KUKA KRL data list: kuka_ros_driver.dat

&ACCESS RVO2
&REL 13769
&PARAM DISKPATH = KRC:\R1\Program\ROS
DEFDAT  KUKA_ROS_DRIVER PUBLIC
EXT  bas (BAS_COMMAND  :IN,REAL  :IN )

GLOBAL INT ROS_InterfaceVersion=2004
; Controls the communication format of the core server communication
; (must match compile of ROS Node.  See #define in kuka_kss_hw_interface.h)
; 1=EKI_COMM_XML, 2=EKI_COMM_BIN
INT ROS_EKI_COMM_MODE=2

INT ROS_Timeout_RLockID=11
INT ROS_Timeout_SLockID=12
GLOBAL INT ROS_RSI_Conn_Flag=115

E6AXIS ROS_Meas_Pos={A1 -106.622528,A2 -31.4800682,A3 -40.7959671,A4 -36.6705093,A5 72.0757370,A6 139.748947,E1 0.0,E2 0.0,E3 0.0,E4 0.0,E5 0.0,E6 0.0}
E6AXIS ROS_Meas_Vel={A1 0.0,A2 0.0,A3 0.0,A4 0.0,A5 0.0,A6 0.0,E1 0.0,E2 0.0,E3 0.0,E4 0.0,E5 0.0,E6 0.0}
E6AXIS ROS_Meas_Torque={A1 0.0,A2 0.0,A3 0.0,A4 0.0,A5 0.0,A6 0.0,E1 0.0,E2 0.0,E3 0.0,E4 0.0,E5 0.0,E6 0.0}

INT ROS_IPOC=747628430
INT IPOC_END=747628432
; Time for next data send, interval (ms) between sends
INT ROS_Interval=20
GLOBAL BOOL ROS_DoSendTrig=TRUE
GLOBAL BOOL ROS_DidInit=FALSE
; Time for next data collect cycle
INT ROS_NextTrigDC=747628450
INT ROS_IntervalDC=20
GLOBAL BOOL ROS_CommFromSPS=TRUE
GLOBAL INT ROS_InterruptRecv=14
GLOBAL INT ROS_InterruptSend=16
INT recv_status=0

; Operation state types
GLOBAL ENUM ROS_OpStateType Unknown,KRL_PTP,RSI4ms_Pos,RSI12ms_Pos,RSI4ms_Vel,RSI12ms_Vel
GLOBAL ENUM ROS_CommandType ROSC_None,ROSC_Init,ROSC_CmdJpos,ROSC_Start,ROSC_Stop,ROSC_Reset,ROSC_DrivesOn,ROSC_DrivesOff,ROSC_Change,ROSC_Heartbeat,ROSC_SInit,ROSC_SInitName,ROSC_SInitMod,ROSC_SInitRobV,ROSC_SjState,ROSC_Sstatus,ROSC_Sackn
GLOBAL STRUC ROS_CommandItem ROS_CommandType type,CHAR IDstr[8],BOOL isRecv
GLOBAL STRUC ROS_Command ROS_CommandType type,INT cmdID,INT dataID,INT t_recv,INT t_exec,INT i_exe
GLOBAL STRUC ROS_PosItem INT cmdIdx,REAL dt,E6AXIS cmdPos
GLOBAL STRUC ROS_OpStateProgAttr ROS_OpStateType type,CHAR IDstr[64],CHAR prgName[64]
GLOBAL STRUC ROS_OpStateItem ROS_OpStateType type,INT t_recv,INT t_active
GLOBAL STRUC ROS_RobStatusType INT statCode,INT mode,eStop,guardStop,drivesPowered,motionPossible,inMotion,inError,errCode,CHAR opState[64]
GLOBAL STRUC ROS_FeatuesType INT EKI,INT RSI,INT MXA
GLOBAL STRUC CircQueue INT size,INT istart,INT iend

DECL ROS_RobStatusType ROS_RobotStatus
DECL ROS_FeatuesType ROS_SupportFeatures

INT OpStateErrCnt=0
INT OpStateChangeStep=0
INT ROS_CurrentOpStateID=1
DECL GLOBAL ROS_OpStateType ROS_CurrentOpState=#KRL_PTP
DECL GLOBAL ROS_OpStateType ROS_RequestedOpState=#KRL_PTP
BOOL ROS_ChangingOpState=FALSE
CHAR ROS_OpStateProg[256]
ROS_OpStateProg[]="ros_krlptp"

DECL ROS_OpStateType temp_PrevOpState=#KRL_PTP
CHAR tempOpState[64]
tempOpState[]="KRL_PTP"
BOOL tempRB=TRUE

DECL ROS_CommandItem ROS_EmptyCommand={type #ROSC_None,IDstr[] "none",isRecv FALSE}
; Registerd command types
INT ROS_NumCommands=16
INT ROS_MaxCommands=20
DECL GLOBAL ROS_CommandItem ROS_CommandTypes[21] ; last item is always none
ROS_CommandTypes[1]={type #ROSC_Init,IDstr[] "Connect-",isRecv TRUE}
ROS_CommandTypes[2]={type #ROSC_CmdJpos,IDstr[] "CmdJpos-",isRecv TRUE}
ROS_CommandTypes[3]={type #ROSC_Start,IDstr[] "Start---",isRecv TRUE}
ROS_CommandTypes[4]={type #ROSC_Stop,IDstr[] "Stop----",isRecv TRUE}
ROS_CommandTypes[5]={type #ROSC_Reset,IDstr[] "Reset---",isRecv TRUE}
ROS_CommandTypes[6]={type #ROSC_DrivesOn,IDstr[] "DriveOn-",isRecv TRUE}
ROS_CommandTypes[7]={type #ROSC_DrivesOff,IDstr[] "DriveOff",isRecv TRUE}
ROS_CommandTypes[8]={type #ROSC_Change,IDstr[] "Change--",isRecv TRUE}
ROS_CommandTypes[9]={type #ROSC_Heartbeat,IDstr[] "HB------",isRecv TRUE}
ROS_CommandTypes[10]={type #ROSC_SInit,IDstr[] "Init----",isRecv FALSE}
ROS_CommandTypes[11]={type #ROSC_SInitName,IDstr[] "InitName",isRecv FALSE}
ROS_CommandTypes[12]={type #ROSC_SInitMod,IDstr[] "InitMod-",isRecv FALSE}
ROS_CommandTypes[13]={type #ROSC_SInitRobV,IDstr[] "InitRobV",isRecv FALSE}
ROS_CommandTypes[14]={type #ROSC_SjState,IDstr[] "JState--",isRecv FALSE}
ROS_CommandTypes[15]={type #ROSC_Sstatus,IDstr[] "Status--",isRecv FALSE}
ROS_CommandTypes[16]={type #ROSC_Sackn,IDstr[] "Ack-----",isRecv FALSE}
ROS_CommandTypes[17]={type #ROSC_None,IDstr[] "none",isRecv FALSE}
ROS_CommandTypes[18]={type #ROSC_None,IDstr[] "none",isRecv FALSE}
ROS_CommandTypes[19]={type #ROSC_None,IDstr[] "none",isRecv FALSE}
ROS_CommandTypes[20]={type #ROSC_None,IDstr[] "none",isRecv FALSE}
ROS_CommandTypes[21]={type #ROSC_None,IDstr[] "none"}
; Quick indexes for send command
GLOBAL INT ROS_Cmd_____Init=10
GLOBAL INT ROS_Cmd_InitName=11
GLOBAL INT ROS_Cmd__InitMod=12
GLOBAL INT ROS_Cmd_InitRobV=13
GLOBAL INT ROS_Cmd___JState=14
GLOBAL INT ROS_Cmd___Status=15
GLOBAL INT ROS_Cmd_____Ackn=16

; This static structure maps between OpState, communication, and KRL program name
INT ROS_NumOpPrograms=6
DECL ROS_OpStateProgAttr ROS_OpPrograms[10]
ROS_OpPrograms[1]={type #KRL_PTP,IDstr[] "KRL_PTP",prgName[] "ros_krlptp"}
ROS_OpPrograms[2]={type #RSI4ms_Pos,IDstr[] "RSI4ms_Pos",prgName[] "ros_rsi_ext"}
ROS_OpPrograms[3]={type #RSI12ms_Pos,IDstr[] "RSI12ms_Pos",prgName[] "ros_rsi_12ms"}
ROS_OpPrograms[4]={type #RSI4ms_Vel,IDstr[] "RSI4ms_Vel",prgName[] "ros_rsi_ext"}
ROS_OpPrograms[5]={type #RSI12ms_Vel,IDstr[] "RSI12ms_Vel",prgName[] "ros_rsi_12ms"}
ROS_OpPrograms[6]={type #Unknown,IDstr[] "Unknown",prgName[] "none"}

; Bit mapping of status code
GLOBAL INT ROSSTAT_T1=1
GLOBAL INT ROSSTAT_T2=2
GLOBAL INT ROSSTAT_AUTO=4
GLOBAL INT ROSSTAT_EXT=8
GLOBAL INT ROSSTAT_Estop=16
GLOBAL INT ROSSTAT_GuardStop=32
GLOBAL INT ROSSTAT_DrivesPwr=64
GLOBAL INT ROSSTAT_MotionPossible=128
GLOBAL INT ROSSTAT_InMotion=256
GLOBAL INT ROSSTAT_KRL_PTP=512
GLOBAL INT ROSSTAT_RSI4ms_Pos=1024
GLOBAL INT ROSSTAT_RSI12ms_Pos=2048
GLOBAL INT ROSSTAT_RSI4ms_Vel=4096
GLOBAL INT ROSSTAT_RSI12ms_Vel=8192
GLOBAL INT ROSSTAT_InError=32768
INT ROSSTAT_Code_ID=1



REAL vel_ratio[12]
vel_ratio[1]=0.233695656
vel_ratio[2]=0.202702701
vel_ratio[3]=0.232432425
vel_ratio[4]=2.12917962E-06
vel_ratio[5]=0.00337662338
vel_ratio[6]=0.134297520
vel_ratio[7]=0.0
vel_ratio[8]=0.0
vel_ratio[9]=0.0
vel_ratio[10]=0.0
vel_ratio[11]=0.0
vel_ratio[12]=0.0

BOOL lock_data_collect=FALSE
BOOL lock_data_read=FALSE

; Test & performance monitoring vars
INT t_DataCollect=35
INT n_DataCollect=17
GLOBAL REAL ROS_DataCollect_cycle=2.05882359

INT t_write=22
INT n_write=7
GLOBAL REAL ROS_write_cycle=0.0
INT dbg_err_idx=10

INT n_lockHoldRead=3300
INT n_lockHoldCollect=7438



DECL ROS_Command emptyCMD={type #ROSC_None,cmdID -1,t_recv 0,t_exec 0}



DECL CircQueue CMDlist_q={size 100,istart 50,iend 50}
DECL ROS_Command CMDlist[100]
CMDlist[1]={type #ROSC_CmdJpos,cmdID 747189637,dataID 97,t_recv 747189704,t_exec 747191325}
CMDlist[2]={type #ROSC_CmdJpos,cmdID 747189664,dataID 98,t_recv 747189730,t_exec 747191409}
CMDlist[3]={type #ROSC_CmdJpos,cmdID 747189692,dataID 99,t_recv 747189757,t_exec 747191493}
CMDlist[4]={type #ROSC_CmdJpos,cmdID 747189720,dataID 100,t_recv 747189784,t_exec 747191577}
CMDlist[5]={type #ROSC_CmdJpos,cmdID 747189747,dataID 1,t_recv 747189812,t_exec 747191661}
CMDlist[6]={type #ROSC_CmdJpos,cmdID 747189774,dataID 2,t_recv 747189840,t_exec 747191745}
CMDlist[7]={type #ROSC_CmdJpos,cmdID 747189800,dataID 3,t_recv 747189870,t_exec 747191829}
CMDlist[8]={type #ROSC_CmdJpos,cmdID 747189829,dataID 4,t_recv 747189898,t_exec 747191925}
CMDlist[9]={type #ROSC_CmdJpos,cmdID 747189858,dataID 5,t_recv 747189923,t_exec 747192009}
CMDlist[10]={type #ROSC_CmdJpos,cmdID 747189887,dataID 6,t_recv 747189950,t_exec 747192093}
CMDlist[11]={type #ROSC_CmdJpos,cmdID 747189913,dataID 7,t_recv 747189975,t_exec 747192177}
CMDlist[12]={type #ROSC_CmdJpos,cmdID 747189940,dataID 8,t_recv 747190023,t_exec 747192273}
CMDlist[13]={type #ROSC_CmdJpos,cmdID 747189965,dataID 9,t_recv 747190030,t_exec 747192357}
CMDlist[14]={type #ROSC_CmdJpos,cmdID 747189992,dataID 10,t_recv 747190059,t_exec 747192441}
CMDlist[15]={type #ROSC_CmdJpos,cmdID 747190012,dataID 11,t_recv 747190087,t_exec 747192537}
CMDlist[16]={type #ROSC_CmdJpos,cmdID 747190049,dataID 12,t_recv 747190114,t_exec 747192621}
CMDlist[17]={type #ROSC_CmdJpos,cmdID 747190076,dataID 13,t_recv 747190141,t_exec 747192705}
CMDlist[18]={type #ROSC_CmdJpos,cmdID 747190104,dataID 14,t_recv 747190168,t_exec 747192789}
CMDlist[19]={type #ROSC_CmdJpos,cmdID 747190131,dataID 15,t_recv 747190195,t_exec 747192873}
CMDlist[20]={type #ROSC_CmdJpos,cmdID 747190158,dataID 16,t_recv 747190225,t_exec 747192957}
CMDlist[21]={type #ROSC_CmdJpos,cmdID 747190185,dataID 17,t_recv 747190251,t_exec 747193053}
CMDlist[22]={type #ROSC_CmdJpos,cmdID 747190214,dataID 18,t_recv 747190280,t_exec 747193137}
CMDlist[23]={type #ROSC_CmdJpos,cmdID 747190241,dataID 19,t_recv 747190307,t_exec 747193233}
CMDlist[24]={type #ROSC_CmdJpos,cmdID 747190269,dataID 20,t_recv 747190351,t_exec 747193329}
CMDlist[25]={type #ROSC_CmdJpos,cmdID 747190297,dataID 21,t_recv 747190358,t_exec 747193425}
CMDlist[26]={type #ROSC_CmdJpos,cmdID 747190324,dataID 22,t_recv 747190392,t_exec 747193521}
CMDlist[27]={type #ROSC_CmdJpos,cmdID 747190368,dataID 23,t_recv 747190429,t_exec 747193617}
CMDlist[28]={type #ROSC_CmdJpos,cmdID 747190403,dataID 24,t_recv 747190465,t_exec 747193713}
CMDlist[29]={type #ROSC_CmdJpos,cmdID 747190438,dataID 25,t_recv 747190501,t_exec 747193809}
CMDlist[30]={type #ROSC_CmdJpos,cmdID 747190475,dataID 26,t_recv 747190534,t_exec 747193905}
CMDlist[31]={type #ROSC_CmdJpos,cmdID 747190510,dataID 27,t_recv 747190567,t_exec 747194013}
CMDlist[32]={type #ROSC_CmdJpos,cmdID 747190544,dataID 28,t_recv 747190603,t_exec 747194133}
CMDlist[33]={type #ROSC_CmdJpos,cmdID 747190578,dataID 29,t_recv 747190640,t_exec 747194241}
CMDlist[34]={type #ROSC_CmdJpos,cmdID 747190614,dataID 30,t_recv 747190676,t_exec 747194361}
CMDlist[35]={type #ROSC_CmdJpos,cmdID 747190650,dataID 31,t_recv 747190712,t_exec 747194481}
CMDlist[36]={type #ROSC_CmdJpos,cmdID 747190687,dataID 32,t_recv 747190747,t_exec 747194601}
CMDlist[37]={type #ROSC_CmdJpos,cmdID 747190723,dataID 33,t_recv 747190780,t_exec 747194733}
CMDlist[38]={type #ROSC_CmdJpos,cmdID 747190757,dataID 34,t_recv 747190816,t_exec 747194853}
CMDlist[39]={type #ROSC_CmdJpos,cmdID 747190790,dataID 35,t_recv 747190852,t_exec 747194973}
CMDlist[40]={type #ROSC_CmdJpos,cmdID 747190825,dataID 36,t_recv 747190888,t_exec 747195093}
CMDlist[41]={type #ROSC_CmdJpos,cmdID 747190862,dataID 37,t_recv 747190923,t_exec 747195201}
CMDlist[42]={type #ROSC_CmdJpos,cmdID 747190897,dataID 38,t_recv 747190957,t_exec 747195321}
CMDlist[43]={type #ROSC_CmdJpos,cmdID 747190932,dataID 39,t_recv 747191020,t_exec 747195417}
CMDlist[44]={type #ROSC_CmdJpos,cmdID 747190967,dataID 40,t_recv 747191027,t_exec 747195513}
CMDlist[45]={type #ROSC_CmdJpos,cmdID 747190992,dataID 41,t_recv 747191064,t_exec 747195597}
CMDlist[46]={type #ROSC_CmdJpos,cmdID 747191038,dataID 42,t_recv 747191100,t_exec 747195681}
CMDlist[47]={type #ROSC_CmdJpos,cmdID 747191074,dataID 43,t_recv 747191135,t_exec 747195753}
CMDlist[48]={type #ROSC_CmdJpos,cmdID 747191110,dataID 44,t_recv 747191171,t_exec 747195837}
CMDlist[49]={type #ROSC_Stop,cmdID 747233232,t_recv 747233291,t_exec 747233305}
CMDlist[50]={type #ROSC_Reset,cmdID 747246081,t_recv 747246134,t_exec 747246143}
CMDlist[51]={type #ROSC_CmdJpos,cmdID 747152086,dataID 47,t_recv 747152148,t_exec 747154473}
CMDlist[52]={type #ROSC_CmdJpos,cmdID 747152112,dataID 48,t_recv 747152173,t_exec 747154533}
CMDlist[53]={type #ROSC_CmdJpos,cmdID 747152138,dataID 49,t_recv 747152202,t_exec 747154605}
CMDlist[54]={type #ROSC_CmdJpos,cmdID 747152163,dataID 50,t_recv 747152231,t_exec 747154653}
CMDlist[55]={type #ROSC_CmdJpos,cmdID 747152190,dataID 51,t_recv 747152261,t_exec 747154713}
CMDlist[56]={type #ROSC_CmdJpos,cmdID 747152220,dataID 52,t_recv 747152290,t_exec 747154773}
CMDlist[57]={type #ROSC_CmdJpos,cmdID 747152249,dataID 53,t_recv 747152317,t_exec 747154821}
CMDlist[58]={type #ROSC_CmdJpos,cmdID 747152278,dataID 54,t_recv 747152343,t_exec 747154857}
CMDlist[59]={type #ROSC_CmdJpos,cmdID 747188462,dataID 55,t_recv 747188514,t_exec 747188516}
CMDlist[60]={type #ROSC_CmdJpos,cmdID 747188491,dataID 56,t_recv 747188546,t_exec 747188548}
CMDlist[61]={type #ROSC_CmdJpos,cmdID 747188523,dataID 57,t_recv 747188579,t_exec 747188582}
CMDlist[62]={type #ROSC_CmdJpos,cmdID 747188555,dataID 58,t_recv 747188613,t_exec 747188733}
CMDlist[63]={type #ROSC_CmdJpos,cmdID 747188588,dataID 59,t_recv 747188650,t_exec 747188757}
CMDlist[64]={type #ROSC_CmdJpos,cmdID 747188625,dataID 60,t_recv 747188684,t_exec 747188781}
CMDlist[65]={type #ROSC_CmdJpos,cmdID 747188659,dataID 61,t_recv 747188716,t_exec 747188817}
CMDlist[66]={type #ROSC_CmdJpos,cmdID 747188693,dataID 62,t_recv 747188749,t_exec 747188853}
CMDlist[67]={type #ROSC_CmdJpos,cmdID 747188725,dataID 63,t_recv 747188790,t_exec 747188889}
CMDlist[68]={type #ROSC_CmdJpos,cmdID 747188759,dataID 64,t_recv 747188797,t_exec 747188937}
CMDlist[69]={type #ROSC_CmdJpos,cmdID 747188759,dataID 65,t_recv 747188826,t_exec 747188985}
CMDlist[70]={type #ROSC_CmdJpos,cmdID 747188780,dataID 66,t_recv 747188857,t_exec 747189033}
CMDlist[71]={type #ROSC_CmdJpos,cmdID 747188815,dataID 67,t_recv 747188884,t_exec 747189093}
CMDlist[72]={type #ROSC_CmdJpos,cmdID 747188846,dataID 68,t_recv 747188911,t_exec 747189153}
CMDlist[73]={type #ROSC_CmdJpos,cmdID 747188874,dataID 69,t_recv 747188936,t_exec 747189213}
CMDlist[74]={type #ROSC_CmdJpos,cmdID 747188901,dataID 70,t_recv 747188962,t_exec 747189273}
CMDlist[75]={type #ROSC_CmdJpos,cmdID 747188926,dataID 71,t_recv 747188989,t_exec 747189333}
CMDlist[76]={type #ROSC_CmdJpos,cmdID 747188952,dataID 72,t_recv 747189018,t_exec 747189405}
CMDlist[77]={type #ROSC_CmdJpos,cmdID 747188978,dataID 73,t_recv 747189046,t_exec 747189477}
CMDlist[78]={type #ROSC_CmdJpos,cmdID 747189007,dataID 74,t_recv 747189075,t_exec 747189537}
CMDlist[79]={type #ROSC_CmdJpos,cmdID 747189036,dataID 75,t_recv 747189103,t_exec 747189609}
CMDlist[80]={type #ROSC_CmdJpos,cmdID 747189063,dataID 76,t_recv 747189130,t_exec 747189681}
CMDlist[81]={type #ROSC_CmdJpos,cmdID 747189092,dataID 77,t_recv 747189155,t_exec 747189753}
CMDlist[82]={type #ROSC_CmdJpos,cmdID 747189119,dataID 78,t_recv 747189181,t_exec 747189825}
CMDlist[83]={type #ROSC_CmdJpos,cmdID 747189145,dataID 79,t_recv 747189211,t_exec 747189899}
CMDlist[84]={type #ROSC_CmdJpos,cmdID 747189171,dataID 80,t_recv 747189238,t_exec 747189969}
CMDlist[85]={type #ROSC_CmdJpos,cmdID 747189199,dataID 81,t_recv 747189266,t_exec 747190053}
CMDlist[86]={type #ROSC_CmdJpos,cmdID 747189227,dataID 82,t_recv 747189294,t_exec 747190125}
CMDlist[87]={type #ROSC_CmdJpos,cmdID 747189254,dataID 83,t_recv 747189323,t_exec 747190197}
CMDlist[88]={type #ROSC_CmdJpos,cmdID 747189282,dataID 84,t_recv 747189350,t_exec 747190281}
CMDlist[89]={type #ROSC_CmdJpos,cmdID 747189311,dataID 85,t_recv 747189377,t_exec 747190353}
CMDlist[90]={type #ROSC_CmdJpos,cmdID 747189340,dataID 86,t_recv 747189404,t_exec 747190425}
CMDlist[91]={type #ROSC_CmdJpos,cmdID 747189367,dataID 87,t_recv 747189431,t_exec 747190509}
CMDlist[92]={type #ROSC_CmdJpos,cmdID 747189392,dataID 88,t_recv 747189459,t_exec 747190593}
CMDlist[93]={type #ROSC_CmdJpos,cmdID 747189420,dataID 89,t_recv 747189486,t_exec 747190677}
CMDlist[94]={type #ROSC_CmdJpos,cmdID 747189448,dataID 90,t_recv 747189514,t_exec 747190749}
CMDlist[95]={type #ROSC_CmdJpos,cmdID 747189475,dataID 91,t_recv 747189541,t_exec 747190833}
CMDlist[96]={type #ROSC_CmdJpos,cmdID 747189503,dataID 92,t_recv 747189566,t_exec 747190917}
CMDlist[97]={type #ROSC_CmdJpos,cmdID 747189530,dataID 93,t_recv 747189591,t_exec 747191001}
CMDlist[98]={type #ROSC_CmdJpos,cmdID 747189556,dataID 94,t_recv 747189621,t_exec 747191073}
CMDlist[99]={type #ROSC_CmdJpos,cmdID 747189581,dataID 95,t_recv 747189648,t_exec 747191157}
CMDlist[100]={type #ROSC_CmdJpos,cmdID 747189609,dataID 96,t_recv 747189676,t_exec 747191241}


GLOBAL E6AXIS g_joint_pos_empty={A1 0.0,A2 0.0,A3 0.0,A4 0.0,A5 0.0,A6 0.0,E1 0.0,E2 0.0,E3 0.0,E4 0.0,E5 0.0,E6 0.0}
GLOBAL E6AXIS ROS_joint_pos_tgt={A1 -106.622528,A2 -31.4800682,A3 -40.7959671,A4 -36.6705093,A5 72.0757370,A6 139.748947,E1 -0.00564089,E2 0.00186683913,E3 0.0,E4 0.0,E5 0.0,E6 0.0}
; Handshake variables to main motion run to avoid running the same point repeatedly
GLOBAL INT ROS_move_ID=747191110
GLOBAL INT ROS_move_ID_previous=387826110
GLOBAL REAL ROS_move_interval=0.0360000
BOOL ROS_move_init=FALSE

BOOL lock_cmdPos_receive=FALSE
BOOL lock_cmdPos_read=FALSE

DECL CircQueue JPosList_q={size 100,istart 44,iend 44}
DECL ROS_PosItem JPos_log[100]
JPos_log[1]={cmdIdx 5,dt 0.0280000,cmdPos {A1 -62.1725273,A2 -55.9574471,A3 7.92842150,A4 15.2566948,A5 9.14249134,A6 139.747818,E1 -0.00282434770,E2 0.000934711075,E3 0.0,E4 0.0,E5 0.0,E6 0.0}}
JPos_log[2]={cmdIdx 6,dt 0.0270000,cmdPos {A1 -63.2651711,A2 -55.3557587,A3 6.73070860,A4 13.9802523,A5 10.6894779,A6 139.747849,E1 -0.00289358222,E2 0.000957624114,E3 0.0,E4 0.0,E5 0.0,E6 0.0}}
JPos_log[3]={cmdIdx 7,dt 0.0270000,cmdPos {A1 -64.3578110,A2 -54.7540703,A3 5.53299570,A4 12.7038097,A5 12.2364635,A6 139.747879,E1 -0.00296281651,E2 0.000980537,E3 0.0,E4 0.0,E5 0.0,E6 0.0}}
JPos_log[4]={cmdIdx 8,dt 0.0260000,cmdPos {A1 -65.4099884,A2 -54.1746674,A3 4.37964249,A4 11.4746428,A5 13.7261543,A6 139.747894,E1 -0.00302948686,E2 0.00100260146,E3 0.0,E4 0.0,E5 0.0,E6 0.0}}
JPos_log[5]={cmdIdx 9,dt 0.0290000,cmdPos {A1 -66.5835648,A2 -53.5284119,A3 3.09321046,A4 10.1036491,A5 15.3877316,A6 139.747925,E1 -0.00310385,E2 0.00102721166,E3 0.0,E4 0.0,E5 0.0,E6 0.0}}
JPos_log[6]={cmdIdx 10,dt 0.0290000,cmdPos {A1 -67.7571487,A2 -52.8821526,A3 1.80677807,A4 8.73265553,A5 17.0493088,A6 139.747955,E1 -0.00317821279,E2 0.00105182198,E3 0.0,E4 0.0,E5 0.0,E6 0.0}}
JPos_log[7]={cmdIdx 11,dt 0.0290000,cmdPos {A1 -68.9307251,A2 -52.2358971,A3 0.520345867,A4 7.36166191,A5 18.7108860,A6 139.747986,E1 -0.00325257587,E2 0.00107643218,E3 0.0,E4 0.0,E5 0.0,E6 0.0}}
JPos_log[8]={cmdIdx 12,dt 0.0260000,cmdPos {A1 -69.9828949,A2 -51.6564941,A3 -0.633007228,A4 6.13249540,A5 20.2005768,A6 139.748016,E1 -0.00331924600,E2 0.00109849661,E3 0.0,E4 0.0,E5 0.0,E6 0.0}}
JPos_log[9]={cmdIdx 13,dt 0.0270000,cmdPos {A1 -71.0755386,A2 -51.0548058,A3 -1.83072007,A4 4.85605288,A5 21.7475624,A6 139.748047,E1 -0.00338848052,E2 0.00112140959,E3 0.0,E4 0.0,E5 0.0,E6 0.0}}
JPos_log[10]={cmdIdx 14,dt 0.0250000,cmdPos {A1 -72.0872498,A2 -50.4976883,A3 -2.93971348,A4 3.67416167,A5 23.1799583,A6 139.748077,E1 -0.00345258671,E2 0.00114262535,E3 0.0,E4 0.0,E5 0.0,E6 0.0}}
JPos_log[11]={cmdIdx 15,dt 0.0270000,cmdPos {A1 -73.1798859,A2 -49.8960,A3 -4.13742638,A4 2.39771938,A5 24.7269440,A6 139.748093,E1 -0.00352182123,E2 0.00116553833,E3 0.0,E4 0.0,E5 0.0,E6 0.0}}
JPos_log[12]={cmdIdx 16,dt 0.0200000,cmdPos {A1 -73.9892502,A2 -49.4503059,A3 -5.02462101,A4 1.45220637,A5 25.8728600,A6 139.748123,E1 -0.00357310590,E2 0.00118251087,E3 0.0,E4 0.0,E5 0.0,E6 0.0}}
JPos_log[13]={cmdIdx 17,dt 0.0370000,cmdPos {A1 -75.4865799,A2 -48.6257706,A3 -6.66593122,A4 -0.296992451,A5 27.9928036,A6 139.748154,E1 -0.00366798276,E2 0.00121391017,E3 0.0,E4 0.0,E5 0.0,E6 0.0}}
JPos_log[14]={cmdIdx 18,dt 0.0270000,cmdPos {A1 -76.5792236,A2 -48.0240822,A3 -7.86364365,A4 -1.57343483,A5 29.5397892,A6 139.748184,E1 -0.00373721728,E2 0.00123682315,E3 0.0,E4 0.0,E5 0.0,E6 0.0}}
JPos_log[15]={cmdIdx 19,dt 0.0280000,cmdPos {A1 -77.7123337,A2 -47.4001083,A3 -9.10571671,A4 -2.89715290,A5 31.1440716,A6 139.748215,E1 -0.00380901620,E2 0.00126058480,E3 0.0,E4 0.0,E5 0.0,E6 0.0}}
JPos_log[16]={cmdIdx 20,dt 0.0270000,cmdPos {A1 -78.8049698,A2 -46.7984200,A3 -10.3034296,A4 -4.17359543,A5 32.6910553,A6 139.748245,E1 -0.00387825072,E2 0.00128349778,E3 0.0,E4 0.0,E5 0.0,E6 0.0}}
JPos_log[17]={cmdIdx 21,dt 0.0270000,cmdPos {A1 -79.8976135,A2 -46.1967316,A3 -11.5011425,A4 -5.45003796,A5 34.2380447,A6 139.748276,E1 -0.00394748524,E2 0.00130641076,E3 0.0,E4 0.0,E5 0.0,E6 0.0}}
JPos_log[18]={cmdIdx 22,dt 0.0270000,cmdPos {A1 -80.9902573,A2 -45.5950470,A3 -12.6988544,A4 -6.72648,A5 35.7850304,A6 139.748291,E1 -0.00401671976,E2 0.00132932374,E3 0.0,E4 0.0,E5 0.0,E6 0.0}}
JPos_log[19]={cmdIdx 23,dt 0.0290000,cmdPos {A1 -82.1638336,A2 -44.9487877,A3 -13.9852867,A4 -8.09747410,A5 37.4466057,A6 139.748322,E1 -0.00409108261,E2 0.00135393406,E3 0.0,E4 0.0,E5 0.0,E6 0.0}}
JPos_log[20]={cmdIdx 24,dt 0.0270000,cmdPos {A1 -83.2564774,A2 -44.3471,A3 -15.1830,A4 -9.37391663,A5 38.9935913,A6 139.748352,E1 -0.00416031713,E2 0.00137684704,E3 0.0,E4 0.0,E5 0.0,E6 0.0}}
JPos_log[21]={cmdIdx 25,dt 0.0280000,cmdPos {A1 -84.3895874,A2 -43.7231293,A3 -16.4250717,A4 -10.6976347,A5 40.5978737,A6 139.748383,E1 -0.00423211604,E2 0.00140060869,E3 0.0,E4 0.0,E5 0.0,E6 0.0}}
JPos_log[22]={cmdIdx 26,dt 0.0280000,cmdPos {A1 -85.5227,A2 -43.0991554,A3 -17.6671448,A4 -12.0213528,A5 42.2021561,A6 139.748413,E1 -0.00430391449,E2 0.00142437033,E3 0.0,E4 0.0,E5 0.0,E6 0.0}}
JPos_log[23]={cmdIdx 27,dt 0.0270000,cmdPos {A1 -86.6153412,A2 -42.4974670,A3 -18.8648586,A4 -13.2977943,A5 43.7491417,A6 139.748444,E1 -0.00437314902,E2 0.00144728331,E3 0.0,E4 0.0,E5 0.0,E6 0.0}}
JPos_log[24]={cmdIdx 28,dt 0.0440000,cmdPos {A1 -88.3959427,A2 -41.5169411,A3 -20.8166866,A4 -15.3779230,A5 46.2701569,A6 139.748489,E1 -0.00448597595,E2 0.00148462295,E3 0.0,E4 0.0,E5 0.0,E6 0.0}}
JPos_log[25]={cmdIdx 29,dt 0.0350000,cmdPos {A1 -89.8123322,A2 -40.7369728,A3 -22.3692760,A4 -17.0325699,A5 48.2755089,A6 139.748520,E1 -0.00457572425,E2 0.00151432503,E3 0.0,E4 0.0,E5 0.0,E6 0.0}}
JPos_log[26]={cmdIdx 30,dt 0.0350000,cmdPos {A1 -91.2287216,A2 -39.9570084,A3 -23.9218674,A4 -18.6872177,A5 50.2808609,A6 139.748550,E1 -0.00466547254,E2 0.00154402701,E3 0.0,E4 0.0,E5 0.0,E6 0.0}}
JPos_log[27]={cmdIdx 31,dt 0.0370000,cmdPos {A1 -92.7260437,A2 -39.1324730,A3 -25.5631771,A4 -20.4364166,A5 52.4008064,A6 139.748596,E1 -0.00476034964,E2 0.00157542631,E3 0.0,E4 0.0,E5 0.0,E6 0.0}}
JPos_log[28]={cmdIdx 32,dt 0.0350000,cmdPos {A1 -94.1424332,A2 -38.3525085,A3 -27.1157684,A4 -22.0910645,A5 54.4061584,A6 139.748627,E1 -0.00485009793,E2 0.00160512840,E3 0.0,E4 0.0,E5 0.0,E6 0.0}}
JPos_log[29]={cmdIdx 33,dt 0.0340000,cmdPos {A1 -95.5351486,A2 -37.5855789,A3 -28.6424103,A4 -23.7180576,A5 56.3779907,A6 139.748672,E1 -0.00493834633,E2 0.00163433398,E3 0.0,E4 0.0,E5 0.0,E6 0.0}}
JPos_log[30]={cmdIdx 34,dt 0.0340000,cmdPos {A1 -96.9221573,A2 -36.8217926,A3 -30.1627922,A4 -25.3383789,A5 58.3417435,A6 139.748703,E1 -0.00502623292,E2 0.00166341977,E3 0.0,E4 0.0,E5 0.0,E6 0.0}}
JPos_log[31]={cmdIdx 35,dt 0.0360000,cmdPos {A1 -98.2725525,A2 -36.0781631,A3 -31.6430511,A4 -26.9159393,A5 60.2536697,A6 139.748734,E1 -0.00511180,E2 0.00169173803,E3 0.0,E4 0.0,E5 0.0,E6 0.0}}
JPos_log[32]={cmdIdx 36,dt 0.0360000,cmdPos {A1 -99.5495300,A2 -35.3749695,A3 -33.0428238,A4 -28.4077244,A5 62.0616417,A6 139.748764,E1 -0.00519271474,E2 0.00171851658,E3 0.0,E4 0.0,E5 0.0,E6 0.0}}
JPos_log[33]={cmdIdx 37,dt 0.0370000,cmdPos {A1 -100.730888,A2 -34.7244301,A3 -34.3377800,A4 -29.7878036,A5 63.7342300,A6 139.748795,E1 -0.00526757073,E2 0.00174329,E3 0.0,E4 0.0,E5 0.0,E6 0.0}}
JPos_log[34]={cmdIdx 38,dt 0.0360000,cmdPos {A1 -101.813744,A2 -34.1281319,A3 -35.5247650,A4 -31.0528107,A5 65.2673569,A6 139.748825,E1 -0.00533618499,E2 0.00176599773,E3 0.0,E4 0.0,E5 0.0,E6 0.0}}
JPos_log[35]={cmdIdx 39,dt 0.0340000,cmdPos {A1 -102.758011,A2 -33.6081467,A3 -36.5598373,A4 -32.1559219,A5 66.6042786,A6 139.748856,E1 -0.00539601827,E2 0.00178579928,E3 0.0,E4 0.0,E5 0.0,E6 0.0}}
JPos_log[36]={cmdIdx 40,dt 0.0330000,cmdPos {A1 -103.485611,A2 -33.2074776,A3 -37.3574028,A4 -33.0059166,A5 67.6344299,A6 139.748871,E1 -0.00544212200,E2 0.00180105725,E3 0.0,E4 0.0,E5 0.0,E6 0.0}}
JPos_log[37]={cmdIdx 41,dt 0.0350000,cmdPos {A1 -104.116714,A2 -32.8599472,A3 -38.0492,A4 -33.7431831,A5 68.5279541,A6 139.748886,E1 -0.00548211113,E2 0.00181429170,E3 0.0,E4 0.0,E5 0.0,E6 0.0}}
JPos_log[38]={cmdIdx 42,dt 0.0370000,cmdPos {A1 -104.720726,A2 -32.5273361,A3 -38.7112923,A4 -34.4488,A5 69.3831329,A6 139.748901,E1 -0.00552038429,E2 0.00182695792,E3 0.0,E4 0.0,E5 0.0,E6 0.0}}
JPos_log[39]={cmdIdx 43,dt 0.0350000,cmdPos {A1 -105.247467,A2 -32.2372742,A3 -39.2886848,A4 -35.0641479,A5 70.1289,A6 139.748917,E1 -0.00555376057,E2 0.00183800387,E3 0.0,E4 0.0,E5 0.0,E6 0.0}}
JPos_log[40]={cmdIdx 44,dt 0.0350000,cmdPos {A1 -105.720406,A2 -31.9768429,A3 -39.8070946,A4 -35.6166344,A5 70.7984924,A6 139.748932,E1 -0.00558372773,E2 0.00184792140,E3 0.0,E4 0.0,E5 0.0,E6 0.0}}
JPos_log[41]={cmdIdx 45,dt 0.0350000,cmdPos {A1 -106.115677,A2 -31.7591763,A3 -40.2403793,A4 -36.0784,A5 71.3581238,A6 139.748932,E1 -0.00560877379,E2 0.00185621041,E3 0.0,E4 0.0,E5 0.0,E6 0.0}}
JPos_log[42]={cmdIdx 46,dt 0.0250000,cmdPos {A1 -106.335602,A2 -31.6380672,A3 -40.4814568,A4 -36.3353233,A5 71.6695,A6 139.748947,E1 -0.00562270964,E2 0.00186082232,E3 0.0,E4 0.0,E5 0.0,E6 0.0}}
JPos_log[43]={cmdIdx 47,dt 0.0460000,cmdPos {A1 -106.578506,A2 -31.5043068,A3 -40.7477188,A4 -36.6190910,A5 72.0134125,A6 139.748947,E1 -0.00563810114,E2 0.00186591607,E3 0.0,E4 0.0,E5 0.0,E6 0.0}}
JPos_log[44]={cmdIdx 48,dt 0.0360000,cmdPos {A1 -106.622528,A2 -31.4800682,A3 -40.7959671,A4 -36.6705093,A5 72.0757370,A6 139.748947,E1 -0.00564089,E2 0.00186683913,E3 0.0,E4 0.0,E5 0.0,E6 0.0}}
JPos_log[45]={cmdIdx 49,dt 0.0260000,cmdPos {A1 -14.3644066,A2 -80.5024490,A3 60.3516808,A4 67.3275833,A5 -53.9648666,A6 139.746643,E1 0.000590378651,E2 -0.00209156843,E3 0.0,E4 0.0,E5 0.0,E6 0.0}}
JPos_log[46]={cmdIdx 50,dt 0.0290000,cmdPos {A1 -15.0494108,A2 -80.5024948,A3 59.5970306,A4 67.3276291,A5 -53.9649277,A6 139.746658,E1 0.000597995764,E2 -0.00211855397,E3 0.0,E4 0.0,E5 0.0,E6 0.0}}
JPos_log[47]={cmdIdx 51,dt 0.0280000,cmdPos {A1 -15.6574450,A2 -80.5025330,A3 58.9271774,A4 67.3276672,A5 -53.9649811,A6 139.746658,E1 0.000604757,E2 -0.00214250735,E3 0.0,E4 0.0,E5 0.0,E6 0.0}}
JPos_log[48]={cmdIdx 52,dt 0.0280000,cmdPos {A1 -16.2008190,A2 -80.5025635,A3 58.3285599,A4 67.3277054,A5 -53.9650269,A6 139.746674,E1 0.000610799179,E2 -0.00216391333,E3 0.0,E4 0.0,E5 0.0,E6 0.0}}
JPos_log[49]={cmdIdx 53,dt 0.0260000,cmdPos {A1 -16.6365185,A2 -80.5025940,A3 57.8485603,A4 67.3277359,A5 -53.9650650,A6 139.746674,E1 0.000615644094,E2 -0.00218107761,E3 0.0,E4 0.0,E5 0.0,E6 0.0}}
JPos_log[50]={cmdIdx 54,dt 0.0260000,cmdPos {A1 -16.9965782,A2 -80.5026169,A3 57.4518929,A4 67.3277588,A5 -53.9651,A6 139.746674,E1 0.000619647850,E2 -0.00219526212,E3 0.0,E4 0.0,E5 0.0,E6 0.0}}
JPos_log[51]={cmdIdx 55,dt 0.0250000,cmdPos {A1 -17.2649841,A2 -80.5026321,A3 57.1562,A4 67.3277740,A5 -53.9651222,A6 139.746674,E1 0.000622632506,E2 -0.00220583589,E3 0.0,E4 0.0,E5 0.0,E6 0.0}}
JPos_log[52]={cmdIdx 56,dt 0.0270000,cmdPos {A1 -17.4654026,A2 -80.5026474,A3 56.9354019,A4 67.3277893,A5 -53.9651375,A6 139.746689,E1 0.000624861103,E2 -0.00221373141,E3 0.0,E4 0.0,E5 0.0,E6 0.0}}
JPos_log[53]={cmdIdx 57,dt 0.0300000,cmdPos {A1 -17.5805531,A2 -80.5026550,A3 56.8085442,A4 67.3278,A5 -53.9651489,A6 139.746689,E1 0.000626141555,E2 -0.00221826765,E3 0.0,E4 0.0,E5 0.0,E6 0.0}}
JPos_log[54]={cmdIdx 58,dt 0.0290000,cmdPos {A1 -17.5993538,A2 -80.5026550,A3 56.7878342,A4 67.3278,A5 -53.9651489,A6 139.746689,E1 0.000626350637,E2 -0.00221900828,E3 0.0,E4 0.0,E5 0.0,E6 0.0}}
JPos_log[55]={cmdIdx 59,dt 0.0310000,cmdPos {A1 -17.6183434,A2 -80.4921951,A3 56.7670174,A4 67.3056183,A5 -53.9382629,A6 139.746689,E1 0.000616256555,E2 -0.00218711211,E3 0.0,E4 0.0,E5 0.0,E6 0.0}}
JPos_log[56]={cmdIdx 60,dt 0.0280000,cmdPos {A1 -17.7043266,A2 -80.4448471,A3 56.6727676,A4 67.2051697,A5 -53.8165283,A6 139.746689,E1 0.000572450052,E2 -0.00204941514,E3 0.0,E4 0.0,E5 0.0,E6 0.0}}
JPos_log[57]={cmdIdx 61,dt 0.0290000,cmdPos {A1 -17.8910942,A2 -80.3420,A3 56.4680405,A4 66.9869843,A5 -53.5520973,A6 139.746689,E1 0.000482904317,E2 -0.00177018612,E3 0.0,E4 0.0,E5 0.0,E6 0.0}}
JPos_log[58]={cmdIdx 62,dt 0.0320000,cmdPos {A1 -18.2141380,A2 -80.1641083,A3 56.1139297,A4 66.6096,A5 -53.0947266,A6 139.746704,E1 0.000341430394,E2 -0.00133472227,E3 0.0,E4 0.0,E5 0.0,E6 0.0}}
JPos_log[59]={cmdIdx 63,dt 0.0320000,cmdPos {A1 -18.6380062,A2 -79.9306946,A3 55.6493034,A4 66.1144257,A5 -52.4946022,A6 139.746719,E1 0.000179555369,E2 -0.000847501564,E3 0.0,E4 0.0,E5 0.0,E6 0.0}}
JPos_log[60]={cmdIdx 64,dt 0.0330000,cmdPos {A1 -19.1446476,A2 -79.6517,A3 55.0939445,A4 65.5225601,A5 -51.7772903,A6 139.746735,E1 2.33041046E-05,E2 -0.000397049676,E3 0.0,E4 0.0,E5 0.0,E6 0.0}}
JPos_log[61]={cmdIdx 65,dt 0.0370000,cmdPos {A1 -19.7553940,A2 -79.3153839,A3 54.4244652,A4 64.8090744,A5 -50.9125824,A6 139.746750,E1 -0.000105858584,E2 -6.37531630E-05,E3 0.0,E4 0.0,E5 0.0,E6 0.0}}
JPos_log[62]={cmdIdx 66,dt 0.0340000,cmdPos {A1 -20.3424530,A2 -78.9921,A3 53.7809525,A4 64.1232681,A5 -50.0814133,A6 139.746765,E1 -0.000172276414,E2 5.20744034E-05,E3 0.0,E4 0.0,E5 0.0,E6 0.0}}
JPos_log[63]={cmdIdx 67,dt 0.0340000,cmdPos {A1 -20.9898243,A2 -78.6356201,A3 53.0713310,A4 63.3669968,A5 -49.1648483,A6 139.746780,E1 -0.000214834727,E2 7.10990425E-05,E3 0.0,E4 0.0,E5 0.0,E6 0.0}}
JPos_log[64]={cmdIdx 68,dt 0.0320000,cmdPos {A1 -21.7620773,A2 -78.2103577,A3 52.2248154,A4 62.4648361,A5 -48.0714760,A6 139.746796,E1 -0.000263768015,E2 8.72933961E-05,E3 0.0,E4 0.0,E5 0.0,E6 0.0}}
JPos_log[65]={cmdIdx 69,dt 0.0340000,cmdPos {A1 -22.7413063,A2 -77.6711273,A3 51.1514206,A4 61.3208847,A5 -46.6850624,A6 139.746826,E1 -0.000325816218,E2 0.000107828098,E3 0.0,E4 0.0,E5 0.0,E6 0.0}}
JPos_log[66]={cmdIdx 70,dt 0.0340000,cmdPos {A1 -23.7676487,A2 -77.1059494,A3 50.0263824,A4 60.1218948,A5 -45.2319450,A6 139.746841,E1 -0.000390849658,E2 0.000129350767,E3 0.0,E4 0.0,E5 0.0,E6 0.0}}
JPos_log[67]={cmdIdx 71,dt 0.0210000,cmdPos {A1 -24.4380360,A2 -76.7367859,A3 49.2915306,A4 59.3387375,A5 -44.2828,A6 139.746857,E1 -0.000433328300,E2 0.000143408965,E3 0.0,E4 0.0,E5 0.0,E6 0.0}}
JPos_log[68]={cmdIdx 72,dt 0.0350000,cmdPos {A1 -25.6592216,A2 -76.0643082,A3 47.9529152,A4 57.9121284,A5 -42.5538177,A6 139.746887,E1 -0.000510707789,E2 0.000169017527,E3 0.0,E4 0.0,E5 0.0,E6 0.0}}
JPos_log[69]={cmdIdx 73,dt 0.0310000,cmdPos {A1 -26.8036633,A2 -75.4341,A3 46.6984215,A4 56.5751724,A5 -40.9334946,A6 139.746918,E1 -0.000583224581,E2 0.000193016778,E3 0.0,E4 0.0,E5 0.0,E6 0.0}}
JPos_log[70]={cmdIdx 74,dt 0.0280000,cmdPos {A1 -27.9015217,A2 -74.8295364,A3 45.4949913,A4 55.2926369,A5 -39.3791237,A6 139.746948,E1 -0.000652789546,E2 0.000216039160,E3 0.0,E4 0.0,E5 0.0,E6 0.0}}
JPos_log[71]={cmdIdx 75,dt 0.0270000,cmdPos {A1 -29.0208912,A2 -74.2131348,A3 44.2679825,A4 53.9849739,A5 -37.7942963,A6 139.746979,E1 -0.000723717618,E2 0.000239512621,E3 0.0,E4 0.0,E5 0.0,E6 0.0}}
JPos_log[72]={cmdIdx 76,dt 0.0250000,cmdPos {A1 -30.0407505,A2 -73.6515274,A3 43.1500511,A4 52.7935562,A5 -36.3503571,A6 139.747009,E1 -0.000788340287,E2 0.000260899338,E3 0.0,E4 0.0,E5 0.0,E6 0.0}}
JPos_log[73]={cmdIdx 77,dt 0.0260000,cmdPos {A1 -31.0929241,A2 -73.0721207,A3 41.9966965,A4 51.5643883,A5 -34.8606682,A6 139.747025,E1 -0.000855010527,E2 0.000282963709,E3 0.0,E4 0.0,E5 0.0,E6 0.0}}
JPos_log[74]={cmdIdx 78,dt 0.0260000,cmdPos {A1 -32.1451,A2 -72.4927139,A3 40.8433456,A4 50.3352242,A5 -33.3709755,A6 139.747055,E1 -0.000921680825,E2 0.000305028050,E3 0.0,E4 0.0,E5 0.0,E6 0.0}}
JPos_log[75]={cmdIdx 79,dt 0.0290000,cmdPos {A1 -33.3186760,A2 -71.8464584,A3 39.5569115,A4 48.9642296,A5 -31.7094,A6 139.747086,E1 -0.000996043789,E2 0.000329638307,E3 0.0,E4 0.0,E5 0.0,E6 0.0}}
JPos_log[76]={cmdIdx 80,dt 0.0290000,cmdPos {A1 -34.4922562,A2 -71.2002,A3 38.2704811,A4 47.5932350,A5 -30.0478210,A6 139.747116,E1 -0.00107040675,E2 0.000354248565,E3 0.0,E4 0.0,E5 0.0,E6 0.0}}
JPos_log[77]={cmdIdx 81,dt 0.0270000,cmdPos {A1 -35.5849,A2 -70.5985184,A3 37.0727654,A4 46.3167915,A5 -28.5008354,A6 139.747147,E1 -0.00113964127,E2 0.000377161574,E3 0.0,E4 0.0,E5 0.0,E6 0.0}}
JPos_log[78]={cmdIdx 82,dt 0.0290000,cmdPos {A1 -36.7584763,A2 -69.9522552,A3 35.7863350,A4 44.9458,A5 -26.8392582,A6 139.747177,E1 -0.00121400424,E2 0.000401771831,E3 0.0,E4 0.0,E5 0.0,E6 0.0}}
JPos_log[79]={cmdIdx 83,dt 0.0270000,cmdPos {A1 -37.8511200,A2 -69.3505707,A3 34.5886230,A4 43.6693573,A5 -25.2922726,A6 139.747208,E1 -0.00128323876,E2 0.000424684811,E3 0.0,E4 0.0,E5 0.0,E6 0.0}}
JPos_log[80]={cmdIdx 84,dt 0.0260000,cmdPos {A1 -38.9032936,A2 -68.7711639,A3 33.4352684,A4 42.4401894,A5 -23.8025818,A6 139.747223,E1 -0.00134990900,E2 0.000446749182,E3 0.0,E4 0.0,E5 0.0,E6 0.0}}
JPos_log[81]={cmdIdx 85,dt 0.0260000,cmdPos {A1 -39.9554672,A2 -68.1917648,A3 32.2819138,A4 41.2110252,A5 -22.3128910,A6 139.747253,E1 -0.00141657935,E2 0.000468813552,E3 0.0,E4 0.0,E5 0.0,E6 0.0}}
JPos_log[82]={cmdIdx 86,dt 0.0280000,cmdPos {A1 -41.0885773,A2 -67.5677948,A3 31.0398426,A4 39.8873062,A5 -20.7086105,A6 139.747284,E1 -0.00148837804,E2 0.000492575171,E3 0.0,E4 0.0,E5 0.0,E6 0.0}}
JPos_log[83]={cmdIdx 87,dt 0.0280000,cmdPos {A1 -42.2216873,A2 -66.9438171,A3 29.7977695,A4 38.5635872,A5 -19.1043282,A6 139.747314,E1 -0.00156017684,E2 0.000516336819,E3 0.0,E4 0.0,E5 0.0,E6 0.0}}
JPos_log[84]={cmdIdx 88,dt 0.0270000,cmdPos {A1 -43.3143311,A2 -66.3421326,A3 28.6000576,A4 37.2871437,A5 -17.5573425,A6 139.747345,E1 -0.00162941136,E2 0.000539249799,E3 0.0,E4 0.0,E5 0.0,E6 0.0}}
JPos_log[85]={cmdIdx 89,dt 0.0280000,cmdPos {A1 -44.4474411,A2 -65.7181625,A3 27.3579845,A4 35.9634285,A5 -15.9530602,A6 139.747375,E1 -0.00170121,E2 0.000563011388,E3 0.0,E4 0.0,E5 0.0,E6 0.0}}
JPos_log[86]={cmdIdx 90,dt 0.0290000,cmdPos {A1 -45.6210213,A2 -65.0719,A3 26.0715523,A4 34.5924339,A5 -14.2914820,A6 139.747406,E1 -0.00177557301,E2 0.000587621646,E3 0.0,E4 0.0,E5 0.0,E6 0.0}}
JPos_log[87]={cmdIdx 91,dt 0.0290000,cmdPos {A1 -46.7945976,A2 -64.4256439,A3 24.7851200,A4 33.2214394,A5 -12.6299047,A6 139.747437,E1 -0.00184993597,E2 0.000612231903,E3 0.0,E4 0.0,E5 0.0,E6 0.0}}
JPos_log[88]={cmdIdx 92,dt 0.0270000,cmdPos {A1 -47.8872414,A2 -63.8239555,A3 23.5874081,A4 31.9449978,A5 -11.0829182,A6 139.747452,E1 -0.00191917049,E2 0.000635144883,E3 0.0,E4 0.0,E5 0.0,E6 0.0}}
JPos_log[89]={cmdIdx 93,dt 0.0250000,cmdPos {A1 -48.8989487,A2 -63.2668381,A3 22.4784145,A4 30.7631054,A5 -9.65052414,A6 139.747482,E1 -0.00198327657,E2 0.000656360644,E3 0.0,E4 0.0,E5 0.0,E6 0.0}}
JPos_log[90]={cmdIdx 94,dt 0.0280000,cmdPos {A1 -50.0320587,A2 -62.6428642,A3 21.2363415,A4 29.4393883,A5 -8.04624271,A6 139.747513,E1 -0.00205507525,E2 0.000680122292,E3 0.0,E4 0.0,E5 0.0,E6 0.0}}
JPos_log[91]={cmdIdx 95,dt 0.0280000,cmdPos {A1 -51.1651688,A2 -62.0188942,A3 19.9942684,A4 28.1156693,A5 -6.44196033,A6 139.747543,E1 -0.00212687417,E2 0.000703883881,E3 0.0,E4 0.0,E5 0.0,E6 0.0}}
JPos_log[92]={cmdIdx 96,dt 0.0270000,cmdPos {A1 -52.2578125,A2 -61.4172058,A3 18.7965565,A4 26.8392277,A5 -4.89497423,A6 139.747574,E1 -0.00219610846,E2 0.000726796861,E3 0.0,E4 0.0,E5 0.0,E6 0.0}}
JPos_log[93]={cmdIdx 97,dt 0.0280000,cmdPos {A1 -53.3909225,A2 -60.7932320,A3 17.5544834,A4 25.5155087,A5 -3.29069257,A6 139.747604,E1 -0.00226790737,E2 0.000750558509,E3 0.0,E4 0.0,E5 0.0,E6 0.0}}
JPos_log[94]={cmdIdx 98,dt 0.0270000,cmdPos {A1 -54.4835625,A2 -60.1915436,A3 16.3567715,A4 24.2390671,A5 -1.74370658,A6 139.747620,E1 -0.00233714189,E2 0.000773471489,E3 0.0,E4 0.0,E5 0.0,E6 0.0}}
JPos_log[95]={cmdIdx 99,dt 0.0260000,cmdPos {A1 -55.5357399,A2 -59.6121407,A3 15.2034178,A4 23.0099010,A5 -0.254016280,A6 139.747650,E1 -0.00240381202,E2 0.000795535860,E3 0.0,E4 0.0,E5 0.0,E6 0.0}}
JPos_log[96]={cmdIdx 100,dt 0.0250000,cmdPos {A1 -56.5474434,A2 -59.0550232,A3 14.0944242,A4 21.8280087,A5 1.17837822,A6 139.747681,E1 -0.00246791821,E2 0.000816751621,E3 0.0,E4 0.0,E5 0.0,E6 0.0}}
JPos_log[97]={cmdIdx 1,dt 0.0280000,cmdPos {A1 -57.6805534,A2 -58.4310532,A3 12.8523521,A4 20.5042915,A5 2.78266,A6 139.747711,E1 -0.00253971689,E2 0.000840513210,E3 0.0,E4 0.0,E5 0.0,E6 0.0}}
JPos_log[98]={cmdIdx 2,dt 0.0280000,cmdPos {A1 -58.8136635,A2 -57.8070793,A3 11.6102791,A4 19.1805725,A5 4.38694191,A6 139.747742,E1 -0.00261151558,E2 0.000864274858,E3 0.0,E4 0.0,E5 0.0,E6 0.0}}
JPos_log[99]={cmdIdx 3,dt 0.0270000,cmdPos {A1 -59.9063072,A2 -57.2053909,A3 10.4125662,A4 17.9041309,A5 5.93392801,A6 139.747757,E1 -0.00268075,E2 0.000887187838,E3 0.0,E4 0.0,E5 0.0,E6 0.0}}
JPos_log[100]={cmdIdx 4,dt 0.0280000,cmdPos {A1 -61.0394173,A2 -56.5814171,A3 9.17049408,A4 16.5804119,A5 7.53821,A6 139.747787,E1 -0.00275254878,E2 0.000910949486,E3 0.0,E4 0.0,E5 0.0,E6 0.0}}

DECL CircQueue JPosSendList_q={size 100,istart 70,iend 70}
DECL ROS_PosItem JPosSend_log[100]
JPosSend_log[1]={cmdIdx 747289096,dt 0.0,cmdPos {A1 -106.622528,A2 -31.4800682,A3 -40.7959671,A4 -36.6705093,A5 72.0757370,A6 139.748947,E1 0.0,E2 0.0,E3 0.0,E4 0.0,E5 0.0,E6 0.0}}
JPosSend_log[2]={cmdIdx 747289118,dt 0.0,cmdPos {A1 -106.622528,A2 -31.4800682,A3 -40.7959671,A4 -36.6705093,A5 72.0757370,A6 139.748947,E1 0.0,E2 0.0,E3 0.0,E4 0.0,E5 0.0,E6 0.0}}
JPosSend_log[3]={cmdIdx 747289140,dt 0.0,cmdPos {A1 -106.622528,A2 -31.4800682,A3 -40.7959671,A4 -36.6705093,A5 72.0757370,A6 139.748947,E1 0.0,E2 0.0,E3 0.0,E4 0.0,E5 0.0,E6 0.0}}
JPosSend_log[4]={cmdIdx 747289162,dt 0.0,cmdPos {A1 -106.622528,A2 -31.4800682,A3 -40.7959671,A4 -36.6705093,A5 72.0757370,A6 139.748947,E1 0.0,E2 0.0,E3 0.0,E4 0.0,E5 0.0,E6 0.0}}
JPosSend_log[5]={cmdIdx 747289184,dt 0.0,cmdPos {A1 -106.622528,A2 -31.4800682,A3 -40.7959671,A4 -36.6705093,A5 72.0757370,A6 139.748947,E1 0.0,E2 0.0,E3 0.0,E4 0.0,E5 0.0,E6 0.0}}
JPosSend_log[6]={cmdIdx 747289206,dt 0.0,cmdPos {A1 -106.622528,A2 -31.4800682,A3 -40.7959671,A4 -36.6705093,A5 72.0757370,A6 139.748947,E1 0.0,E2 0.0,E3 0.0,E4 0.0,E5 0.0,E6 0.0}}
JPosSend_log[7]={cmdIdx 747289228,dt 0.0,cmdPos {A1 -106.622528,A2 -31.4800682,A3 -40.7959671,A4 -36.6705093,A5 72.0757370,A6 139.748947,E1 0.0,E2 0.0,E3 0.0,E4 0.0,E5 0.0,E6 0.0}}
JPosSend_log[8]={cmdIdx 747289250,dt 0.0,cmdPos {A1 -106.622528,A2 -31.4800682,A3 -40.7959671,A4 -36.6705093,A5 72.0757370,A6 139.748947,E1 0.0,E2 0.0,E3 0.0,E4 0.0,E5 0.0,E6 0.0}}
JPosSend_log[9]={cmdIdx 747289272,dt 0.0,cmdPos {A1 -106.622528,A2 -31.4800682,A3 -40.7959671,A4 -36.6705093,A5 72.0757370,A6 139.748947,E1 0.0,E2 0.0,E3 0.0,E4 0.0,E5 0.0,E6 0.0}}
JPosSend_log[10]={cmdIdx 747289294,dt 0.0,cmdPos {A1 -106.622528,A2 -31.4800682,A3 -40.7959671,A4 -36.6705093,A5 72.0757370,A6 139.748947,E1 0.0,E2 0.0,E3 0.0,E4 0.0,E5 0.0,E6 0.0}}
JPosSend_log[11]={cmdIdx 747289316,dt 0.0,cmdPos {A1 -106.622528,A2 -31.4800682,A3 -40.7959671,A4 -36.6705093,A5 72.0757370,A6 139.748947,E1 0.0,E2 0.0,E3 0.0,E4 0.0,E5 0.0,E6 0.0}}
JPosSend_log[12]={cmdIdx 747289338,dt 0.0,cmdPos {A1 -106.622528,A2 -31.4800682,A3 -40.7959671,A4 -36.6705093,A5 72.0757370,A6 139.748947,E1 0.0,E2 0.0,E3 0.0,E4 0.0,E5 0.0,E6 0.0}}
JPosSend_log[13]={cmdIdx 747289361,dt 0.0,cmdPos {A1 -106.622528,A2 -31.4800682,A3 -40.7959671,A4 -36.6705093,A5 72.0757370,A6 139.748947,E1 0.0,E2 0.0,E3 0.0,E4 0.0,E5 0.0,E6 0.0}}
JPosSend_log[14]={cmdIdx 747289382,dt 0.0,cmdPos {A1 -106.622528,A2 -31.4800682,A3 -40.7959671,A4 -36.6705093,A5 72.0757370,A6 139.748947,E1 0.0,E2 0.0,E3 0.0,E4 0.0,E5 0.0,E6 0.0}}
JPosSend_log[15]={cmdIdx 747289404,dt 0.0,cmdPos {A1 -106.622528,A2 -31.4800682,A3 -40.7959671,A4 -36.6705093,A5 72.0757370,A6 139.748947,E1 0.0,E2 0.0,E3 0.0,E4 0.0,E5 0.0,E6 0.0}}
JPosSend_log[16]={cmdIdx 747289426,dt 0.0,cmdPos {A1 -106.622528,A2 -31.4800682,A3 -40.7959671,A4 -36.6705093,A5 72.0757370,A6 139.748947,E1 0.0,E2 0.0,E3 0.0,E4 0.0,E5 0.0,E6 0.0}}
JPosSend_log[17]={cmdIdx 747289448,dt 0.0,cmdPos {A1 -106.622528,A2 -31.4800682,A3 -40.7959671,A4 -36.6705093,A5 72.0757370,A6 139.748947,E1 0.0,E2 0.0,E3 0.0,E4 0.0,E5 0.0,E6 0.0}}
JPosSend_log[18]={cmdIdx 747289470,dt 0.0,cmdPos {A1 -106.622528,A2 -31.4800682,A3 -40.7959671,A4 -36.6705093,A5 72.0757370,A6 139.748947,E1 0.0,E2 0.0,E3 0.0,E4 0.0,E5 0.0,E6 0.0}}
JPosSend_log[19]={cmdIdx 747289492,dt 0.0,cmdPos {A1 -106.622528,A2 -31.4800682,A3 -40.7959671,A4 -36.6705093,A5 72.0757370,A6 139.748947,E1 0.0,E2 0.0,E3 0.0,E4 0.0,E5 0.0,E6 0.0}}
JPosSend_log[20]={cmdIdx 747289514,dt 0.0,cmdPos {A1 -106.622528,A2 -31.4800682,A3 -40.7959671,A4 -36.6705093,A5 72.0757370,A6 139.748947,E1 0.0,E2 0.0,E3 0.0,E4 0.0,E5 0.0,E6 0.0}}
JPosSend_log[21]={cmdIdx 747289536,dt 0.0,cmdPos {A1 -106.622528,A2 -31.4800682,A3 -40.7959671,A4 -36.6705093,A5 72.0757370,A6 139.748947,E1 0.0,E2 0.0,E3 0.0,E4 0.0,E5 0.0,E6 0.0}}
JPosSend_log[22]={cmdIdx 747289558,dt 0.0,cmdPos {A1 -106.622528,A2 -31.4800682,A3 -40.7959671,A4 -36.6705093,A5 72.0757370,A6 139.748947,E1 0.0,E2 0.0,E3 0.0,E4 0.0,E5 0.0,E6 0.0}}
JPosSend_log[23]={cmdIdx 747289580,dt 0.0,cmdPos {A1 -106.622528,A2 -31.4800682,A3 -40.7959671,A4 -36.6705093,A5 72.0757370,A6 139.748947,E1 0.0,E2 0.0,E3 0.0,E4 0.0,E5 0.0,E6 0.0}}
JPosSend_log[24]={cmdIdx 747289602,dt 0.0,cmdPos {A1 -106.622528,A2 -31.4800682,A3 -40.7959671,A4 -36.6705093,A5 72.0757370,A6 139.748947,E1 0.0,E2 0.0,E3 0.0,E4 0.0,E5 0.0,E6 0.0}}
JPosSend_log[25]={cmdIdx 747289624,dt 0.0,cmdPos {A1 -106.622528,A2 -31.4800682,A3 -40.7959671,A4 -36.6705093,A5 72.0757370,A6 139.748947,E1 0.0,E2 0.0,E3 0.0,E4 0.0,E5 0.0,E6 0.0}}
JPosSend_log[26]={cmdIdx 747289646,dt 0.0,cmdPos {A1 -106.622528,A2 -31.4800682,A3 -40.7959671,A4 -36.6705093,A5 72.0757370,A6 139.748947,E1 0.0,E2 0.0,E3 0.0,E4 0.0,E5 0.0,E6 0.0}}
JPosSend_log[27]={cmdIdx 747289668,dt 0.0,cmdPos {A1 -106.622528,A2 -31.4800682,A3 -40.7959671,A4 -36.6705093,A5 72.0757370,A6 139.748947,E1 0.0,E2 0.0,E3 0.0,E4 0.0,E5 0.0,E6 0.0}}
JPosSend_log[28]={cmdIdx 747289692,dt 0.0,cmdPos {A1 -106.622528,A2 -31.4800682,A3 -40.7959671,A4 -36.6705093,A5 72.0757370,A6 139.748947,E1 0.0,E2 0.0,E3 0.0,E4 0.0,E5 0.0,E6 0.0}}
JPosSend_log[29]={cmdIdx 747289714,dt 0.0,cmdPos {A1 -106.622528,A2 -31.4800682,A3 -40.7959671,A4 -36.6705093,A5 72.0757370,A6 139.748947,E1 0.0,E2 0.0,E3 0.0,E4 0.0,E5 0.0,E6 0.0}}
JPosSend_log[30]={cmdIdx 747289736,dt 0.0,cmdPos {A1 -106.622528,A2 -31.4800682,A3 -40.7959671,A4 -36.6705093,A5 72.0757370,A6 139.748947,E1 0.0,E2 0.0,E3 0.0,E4 0.0,E5 0.0,E6 0.0}}
JPosSend_log[31]={cmdIdx 747289758,dt 0.0,cmdPos {A1 -106.622528,A2 -31.4800682,A3 -40.7959671,A4 -36.6705093,A5 72.0757370,A6 139.748947,E1 0.0,E2 0.0,E3 0.0,E4 0.0,E5 0.0,E6 0.0}}
JPosSend_log[32]={cmdIdx 747289780,dt 0.0,cmdPos {A1 -106.622528,A2 -31.4800682,A3 -40.7959671,A4 -36.6705093,A5 72.0757370,A6 139.748947,E1 0.0,E2 0.0,E3 0.0,E4 0.0,E5 0.0,E6 0.0}}
JPosSend_log[33]={cmdIdx 747289802,dt 0.0,cmdPos {A1 -106.622528,A2 -31.4800682,A3 -40.7959671,A4 -36.6705093,A5 72.0757370,A6 139.748947,E1 0.0,E2 0.0,E3 0.0,E4 0.0,E5 0.0,E6 0.0}}
JPosSend_log[34]={cmdIdx 747289824,dt 0.0,cmdPos {A1 -106.622528,A2 -31.4800682,A3 -40.7959671,A4 -36.6705093,A5 72.0757370,A6 139.748947,E1 0.0,E2 0.0,E3 0.0,E4 0.0,E5 0.0,E6 0.0}}
JPosSend_log[35]={cmdIdx 747289848,dt 0.0,cmdPos {A1 -106.622528,A2 -31.4800682,A3 -40.7959671,A4 -36.6705093,A5 72.0757370,A6 139.748947,E1 0.0,E2 0.0,E3 0.0,E4 0.0,E5 0.0,E6 0.0}}
JPosSend_log[36]={cmdIdx 747289870,dt 0.0,cmdPos {A1 -106.622528,A2 -31.4800682,A3 -40.7959671,A4 -36.6705093,A5 72.0757370,A6 139.748947,E1 0.0,E2 0.0,E3 0.0,E4 0.0,E5 0.0,E6 0.0}}
JPosSend_log[37]={cmdIdx 747289892,dt 0.0,cmdPos {A1 -106.622528,A2 -31.4800682,A3 -40.7959671,A4 -36.6705093,A5 72.0757370,A6 139.748947,E1 0.0,E2 0.0,E3 0.0,E4 0.0,E5 0.0,E6 0.0}}
JPosSend_log[38]={cmdIdx 747289914,dt 0.0,cmdPos {A1 -106.622528,A2 -31.4800682,A3 -40.7959671,A4 -36.6705093,A5 72.0757370,A6 139.748947,E1 0.0,E2 0.0,E3 0.0,E4 0.0,E5 0.0,E6 0.0}}
JPosSend_log[39]={cmdIdx 747289936,dt 0.0,cmdPos {A1 -106.622528,A2 -31.4800682,A3 -40.7959671,A4 -36.6705093,A5 72.0757370,A6 139.748947,E1 0.0,E2 0.0,E3 0.0,E4 0.0,E5 0.0,E6 0.0}}
JPosSend_log[40]={cmdIdx 747289958,dt 0.0,cmdPos {A1 -106.622528,A2 -31.4800682,A3 -40.7959671,A4 -36.6705093,A5 72.0757370,A6 139.748947,E1 0.0,E2 0.0,E3 0.0,E4 0.0,E5 0.0,E6 0.0}}
JPosSend_log[41]={cmdIdx 747289980,dt 0.0,cmdPos {A1 -106.622528,A2 -31.4800682,A3 -40.7959671,A4 -36.6705093,A5 72.0757370,A6 139.748947,E1 0.0,E2 0.0,E3 0.0,E4 0.0,E5 0.0,E6 0.0}}
JPosSend_log[42]={cmdIdx 747290002,dt 0.0,cmdPos {A1 -106.622528,A2 -31.4800682,A3 -40.7959671,A4 -36.6705093,A5 72.0757370,A6 139.748947,E1 0.0,E2 0.0,E3 0.0,E4 0.0,E5 0.0,E6 0.0}}
JPosSend_log[43]={cmdIdx 747290024,dt 0.0,cmdPos {A1 -106.622528,A2 -31.4800682,A3 -40.7959671,A4 -36.6705093,A5 72.0757370,A6 139.748947,E1 0.0,E2 0.0,E3 0.0,E4 0.0,E5 0.0,E6 0.0}}
JPosSend_log[44]={cmdIdx 747290046,dt 0.0,cmdPos {A1 -106.622528,A2 -31.4800682,A3 -40.7959671,A4 -36.6705093,A5 72.0757370,A6 139.748947,E1 0.0,E2 0.0,E3 0.0,E4 0.0,E5 0.0,E6 0.0}}
JPosSend_log[45]={cmdIdx 747290068,dt 0.0,cmdPos {A1 -106.622528,A2 -31.4800682,A3 -40.7959671,A4 -36.6705093,A5 72.0757370,A6 139.748947,E1 0.0,E2 0.0,E3 0.0,E4 0.0,E5 0.0,E6 0.0}}
JPosSend_log[46]={cmdIdx 747290091,dt 0.0,cmdPos {A1 -106.622528,A2 -31.4800682,A3 -40.7959671,A4 -36.6705093,A5 72.0757370,A6 139.748947,E1 0.0,E2 0.0,E3 0.0,E4 0.0,E5 0.0,E6 0.0}}
JPosSend_log[47]={cmdIdx 747290113,dt 0.0,cmdPos {A1 -106.622528,A2 -31.4800682,A3 -40.7959671,A4 -36.6705093,A5 72.0757370,A6 139.748947,E1 0.0,E2 0.0,E3 0.0,E4 0.0,E5 0.0,E6 0.0}}
JPosSend_log[48]={cmdIdx 747290135,dt 0.0,cmdPos {A1 -106.622528,A2 -31.4800682,A3 -40.7959671,A4 -36.6705093,A5 72.0757370,A6 139.748947,E1 0.0,E2 0.0,E3 0.0,E4 0.0,E5 0.0,E6 0.0}}
JPosSend_log[49]={cmdIdx 747290157,dt 0.0,cmdPos {A1 -106.622528,A2 -31.4800682,A3 -40.7959671,A4 -36.6705093,A5 72.0757370,A6 139.748947,E1 0.0,E2 0.0,E3 0.0,E4 0.0,E5 0.0,E6 0.0}}
JPosSend_log[50]={cmdIdx 747290179,dt 0.0,cmdPos {A1 -106.622528,A2 -31.4800682,A3 -40.7959671,A4 -36.6705093,A5 72.0757370,A6 139.748947,E1 0.0,E2 0.0,E3 0.0,E4 0.0,E5 0.0,E6 0.0}}
JPosSend_log[51]={cmdIdx 747290201,dt 0.0,cmdPos {A1 -106.622528,A2 -31.4800682,A3 -40.7959671,A4 -36.6705093,A5 72.0757370,A6 139.748947,E1 0.0,E2 0.0,E3 0.0,E4 0.0,E5 0.0,E6 0.0}}
JPosSend_log[52]={cmdIdx 747290223,dt 0.0,cmdPos {A1 -106.622528,A2 -31.4800682,A3 -40.7959671,A4 -36.6705093,A5 72.0757370,A6 139.748947,E1 0.0,E2 0.0,E3 0.0,E4 0.0,E5 0.0,E6 0.0}}
JPosSend_log[53]={cmdIdx 747290245,dt 0.0,cmdPos {A1 -106.622528,A2 -31.4800682,A3 -40.7959671,A4 -36.6705093,A5 72.0757370,A6 139.748947,E1 0.0,E2 0.0,E3 0.0,E4 0.0,E5 0.0,E6 0.0}}
JPosSend_log[54]={cmdIdx 747290267,dt 0.0,cmdPos {A1 -106.622528,A2 -31.4800682,A3 -40.7959671,A4 -36.6705093,A5 72.0757370,A6 139.748947,E1 0.0,E2 0.0,E3 0.0,E4 0.0,E5 0.0,E6 0.0}}
JPosSend_log[55]={cmdIdx 747290289,dt 0.0,cmdPos {A1 -106.622528,A2 -31.4800682,A3 -40.7959671,A4 -36.6705093,A5 72.0757370,A6 139.748947,E1 0.0,E2 0.0,E3 0.0,E4 0.0,E5 0.0,E6 0.0}}
JPosSend_log[56]={cmdIdx 747290311,dt 0.0,cmdPos {A1 -106.622528,A2 -31.4800682,A3 -40.7959671,A4 -36.6705093,A5 72.0757370,A6 139.748947,E1 0.0,E2 0.0,E3 0.0,E4 0.0,E5 0.0,E6 0.0}}
JPosSend_log[57]={cmdIdx 747290333,dt 0.0,cmdPos {A1 -106.622528,A2 -31.4800682,A3 -40.7959671,A4 -36.6705093,A5 72.0757370,A6 139.748947,E1 0.0,E2 0.0,E3 0.0,E4 0.0,E5 0.0,E6 0.0}}
JPosSend_log[58]={cmdIdx 747290355,dt 0.0,cmdPos {A1 -106.622528,A2 -31.4800682,A3 -40.7959671,A4 -36.6705093,A5 72.0757370,A6 139.748947,E1 0.0,E2 0.0,E3 0.0,E4 0.0,E5 0.0,E6 0.0}}
JPosSend_log[59]={cmdIdx 747290378,dt 0.0,cmdPos {A1 -106.622528,A2 -31.4800682,A3 -40.7959671,A4 -36.6705093,A5 72.0757370,A6 139.748947,E1 0.0,E2 0.0,E3 0.0,E4 0.0,E5 0.0,E6 0.0}}
JPosSend_log[60]={cmdIdx 747290400,dt 0.0,cmdPos {A1 -106.622528,A2 -31.4800682,A3 -40.7959671,A4 -36.6705093,A5 72.0757370,A6 139.748947,E1 0.0,E2 0.0,E3 0.0,E4 0.0,E5 0.0,E6 0.0}}
JPosSend_log[61]={cmdIdx 747290422,dt 0.0,cmdPos {A1 -106.622528,A2 -31.4800682,A3 -40.7959671,A4 -36.6705093,A5 72.0757370,A6 139.748947,E1 0.0,E2 0.0,E3 0.0,E4 0.0,E5 0.0,E6 0.0}}
JPosSend_log[62]={cmdIdx 747290444,dt 0.0,cmdPos {A1 -106.622528,A2 -31.4800682,A3 -40.7959671,A4 -36.6705093,A5 72.0757370,A6 139.748947,E1 0.0,E2 0.0,E3 0.0,E4 0.0,E5 0.0,E6 0.0}}
JPosSend_log[63]={cmdIdx 747290466,dt 0.0,cmdPos {A1 -106.622528,A2 -31.4800682,A3 -40.7959671,A4 -36.6705093,A5 72.0757370,A6 139.748947,E1 0.0,E2 0.0,E3 0.0,E4 0.0,E5 0.0,E6 0.0}}
JPosSend_log[64]={cmdIdx 747290487,dt 0.0,cmdPos {A1 -106.622528,A2 -31.4800682,A3 -40.7959671,A4 -36.6705093,A5 72.0757370,A6 139.748947,E1 0.0,E2 0.0,E3 0.0,E4 0.0,E5 0.0,E6 0.0}}
JPosSend_log[65]={cmdIdx 747290509,dt 0.0,cmdPos {A1 -106.622528,A2 -31.4800682,A3 -40.7959671,A4 -36.6705093,A5 72.0757370,A6 139.748947,E1 0.0,E2 0.0,E3 0.0,E4 0.0,E5 0.0,E6 0.0}}
JPosSend_log[66]={cmdIdx 747290531,dt 0.0,cmdPos {A1 -106.622528,A2 -31.4800682,A3 -40.7959671,A4 -36.6705093,A5 72.0757370,A6 139.748947,E1 0.0,E2 0.0,E3 0.0,E4 0.0,E5 0.0,E6 0.0}}
JPosSend_log[67]={cmdIdx 747290554,dt 0.0,cmdPos {A1 -106.622528,A2 -31.4800682,A3 -40.7959671,A4 -36.6705093,A5 72.0757370,A6 139.748947,E1 0.0,E2 0.0,E3 0.0,E4 0.0,E5 0.0,E6 0.0}}
JPosSend_log[68]={cmdIdx 747290576,dt 0.0,cmdPos {A1 -106.622528,A2 -31.4800682,A3 -40.7959671,A4 -36.6705093,A5 72.0757370,A6 139.748947,E1 0.0,E2 0.0,E3 0.0,E4 0.0,E5 0.0,E6 0.0}}
JPosSend_log[69]={cmdIdx 747290598,dt 0.0,cmdPos {A1 -106.622528,A2 -31.4800682,A3 -40.7959671,A4 -36.6705093,A5 72.0757370,A6 139.748947,E1 0.0,E2 0.0,E3 0.0,E4 0.0,E5 0.0,E6 0.0}}
JPosSend_log[70]={cmdIdx 747290620,dt 0.0,cmdPos {A1 -106.622528,A2 -31.4800682,A3 -40.7959671,A4 -36.6705093,A5 72.0757370,A6 139.748947,E1 0.0,E2 0.0,E3 0.0,E4 0.0,E5 0.0,E6 0.0}}
JPosSend_log[71]={cmdIdx 747288436,dt 0.0,cmdPos {A1 -106.622528,A2 -31.4800682,A3 -40.7959671,A4 -36.6705093,A5 72.0757370,A6 139.748947,E1 0.0,E2 0.0,E3 0.0,E4 0.0,E5 0.0,E6 0.0}}
JPosSend_log[72]={cmdIdx 747288458,dt 0.0,cmdPos {A1 -106.622528,A2 -31.4800682,A3 -40.7959671,A4 -36.6705093,A5 72.0757370,A6 139.748947,E1 0.0,E2 0.0,E3 0.0,E4 0.0,E5 0.0,E6 0.0}}
JPosSend_log[73]={cmdIdx 747288479,dt 0.0,cmdPos {A1 -106.622528,A2 -31.4800682,A3 -40.7959671,A4 -36.6705093,A5 72.0757370,A6 139.748947,E1 0.0,E2 0.0,E3 0.0,E4 0.0,E5 0.0,E6 0.0}}
JPosSend_log[74]={cmdIdx 747288501,dt 0.0,cmdPos {A1 -106.622528,A2 -31.4800682,A3 -40.7959671,A4 -36.6705093,A5 72.0757370,A6 139.748947,E1 0.0,E2 0.0,E3 0.0,E4 0.0,E5 0.0,E6 0.0}}
JPosSend_log[75]={cmdIdx 747288523,dt 0.0,cmdPos {A1 -106.622528,A2 -31.4800682,A3 -40.7959671,A4 -36.6705093,A5 72.0757370,A6 139.748947,E1 0.0,E2 0.0,E3 0.0,E4 0.0,E5 0.0,E6 0.0}}
JPosSend_log[76]={cmdIdx 747288546,dt 0.0,cmdPos {A1 -106.622528,A2 -31.4800682,A3 -40.7959671,A4 -36.6705093,A5 72.0757370,A6 139.748947,E1 0.0,E2 0.0,E3 0.0,E4 0.0,E5 0.0,E6 0.0}}
JPosSend_log[77]={cmdIdx 747288568,dt 0.0,cmdPos {A1 -106.622528,A2 -31.4800682,A3 -40.7959671,A4 -36.6705093,A5 72.0757370,A6 139.748947,E1 0.0,E2 0.0,E3 0.0,E4 0.0,E5 0.0,E6 0.0}}
JPosSend_log[78]={cmdIdx 747288590,dt 0.0,cmdPos {A1 -106.622528,A2 -31.4800682,A3 -40.7959671,A4 -36.6705093,A5 72.0757370,A6 139.748947,E1 0.0,E2 0.0,E3 0.0,E4 0.0,E5 0.0,E6 0.0}}
JPosSend_log[79]={cmdIdx 747288611,dt 0.0,cmdPos {A1 -106.622528,A2 -31.4800682,A3 -40.7959671,A4 -36.6705093,A5 72.0757370,A6 139.748947,E1 0.0,E2 0.0,E3 0.0,E4 0.0,E5 0.0,E6 0.0}}
JPosSend_log[80]={cmdIdx 747288634,dt 0.0,cmdPos {A1 -106.622528,A2 -31.4800682,A3 -40.7959671,A4 -36.6705093,A5 72.0757370,A6 139.748947,E1 0.0,E2 0.0,E3 0.0,E4 0.0,E5 0.0,E6 0.0}}
JPosSend_log[81]={cmdIdx 747288655,dt 0.0,cmdPos {A1 -106.622528,A2 -31.4800682,A3 -40.7959671,A4 -36.6705093,A5 72.0757370,A6 139.748947,E1 0.0,E2 0.0,E3 0.0,E4 0.0,E5 0.0,E6 0.0}}
JPosSend_log[82]={cmdIdx 747288677,dt 0.0,cmdPos {A1 -106.622528,A2 -31.4800682,A3 -40.7959671,A4 -36.6705093,A5 72.0757370,A6 139.748947,E1 0.0,E2 0.0,E3 0.0,E4 0.0,E5 0.0,E6 0.0}}
JPosSend_log[83]={cmdIdx 747288699,dt 0.0,cmdPos {A1 -106.622528,A2 -31.4800682,A3 -40.7959671,A4 -36.6705093,A5 72.0757370,A6 139.748947,E1 0.0,E2 0.0,E3 0.0,E4 0.0,E5 0.0,E6 0.0}}
JPosSend_log[84]={cmdIdx 747288721,dt 0.0,cmdPos {A1 -106.622528,A2 -31.4800682,A3 -40.7959671,A4 -36.6705093,A5 72.0757370,A6 139.748947,E1 0.0,E2 0.0,E3 0.0,E4 0.0,E5 0.0,E6 0.0}}
JPosSend_log[85]={cmdIdx 747288743,dt 0.0,cmdPos {A1 -106.622528,A2 -31.4800682,A3 -40.7959671,A4 -36.6705093,A5 72.0757370,A6 139.748947,E1 0.0,E2 0.0,E3 0.0,E4 0.0,E5 0.0,E6 0.0}}
JPosSend_log[86]={cmdIdx 747288765,dt 0.0,cmdPos {A1 -106.622528,A2 -31.4800682,A3 -40.7959671,A4 -36.6705093,A5 72.0757370,A6 139.748947,E1 0.0,E2 0.0,E3 0.0,E4 0.0,E5 0.0,E6 0.0}}
JPosSend_log[87]={cmdIdx 747288787,dt 0.0,cmdPos {A1 -106.622528,A2 -31.4800682,A3 -40.7959671,A4 -36.6705093,A5 72.0757370,A6 139.748947,E1 0.0,E2 0.0,E3 0.0,E4 0.0,E5 0.0,E6 0.0}}
JPosSend_log[88]={cmdIdx 747288809,dt 0.0,cmdPos {A1 -106.622528,A2 -31.4800682,A3 -40.7959671,A4 -36.6705093,A5 72.0757370,A6 139.748947,E1 0.0,E2 0.0,E3 0.0,E4 0.0,E5 0.0,E6 0.0}}
JPosSend_log[89]={cmdIdx 747288831,dt 0.0,cmdPos {A1 -106.622528,A2 -31.4800682,A3 -40.7959671,A4 -36.6705093,A5 72.0757370,A6 139.748947,E1 0.0,E2 0.0,E3 0.0,E4 0.0,E5 0.0,E6 0.0}}
JPosSend_log[90]={cmdIdx 747288853,dt 0.0,cmdPos {A1 -106.622528,A2 -31.4800682,A3 -40.7959671,A4 -36.6705093,A5 72.0757370,A6 139.748947,E1 0.0,E2 0.0,E3 0.0,E4 0.0,E5 0.0,E6 0.0}}
JPosSend_log[91]={cmdIdx 747288876,dt 0.0,cmdPos {A1 -106.622528,A2 -31.4800682,A3 -40.7959671,A4 -36.6705093,A5 72.0757370,A6 139.748947,E1 0.0,E2 0.0,E3 0.0,E4 0.0,E5 0.0,E6 0.0}}
JPosSend_log[92]={cmdIdx 747288897,dt 0.0,cmdPos {A1 -106.622528,A2 -31.4800682,A3 -40.7959671,A4 -36.6705093,A5 72.0757370,A6 139.748947,E1 0.0,E2 0.0,E3 0.0,E4 0.0,E5 0.0,E6 0.0}}
JPosSend_log[93]={cmdIdx 747288919,dt 0.0,cmdPos {A1 -106.622528,A2 -31.4800682,A3 -40.7959671,A4 -36.6705093,A5 72.0757370,A6 139.748947,E1 0.0,E2 0.0,E3 0.0,E4 0.0,E5 0.0,E6 0.0}}
JPosSend_log[94]={cmdIdx 747288942,dt 0.0,cmdPos {A1 -106.622528,A2 -31.4800682,A3 -40.7959671,A4 -36.6705093,A5 72.0757370,A6 139.748947,E1 0.0,E2 0.0,E3 0.0,E4 0.0,E5 0.0,E6 0.0}}
JPosSend_log[95]={cmdIdx 747288964,dt 0.0,cmdPos {A1 -106.622528,A2 -31.4800682,A3 -40.7959671,A4 -36.6705093,A5 72.0757370,A6 139.748947,E1 0.0,E2 0.0,E3 0.0,E4 0.0,E5 0.0,E6 0.0}}
JPosSend_log[96]={cmdIdx 747288986,dt 0.0,cmdPos {A1 -106.622528,A2 -31.4800682,A3 -40.7959671,A4 -36.6705093,A5 72.0757370,A6 139.748947,E1 0.0,E2 0.0,E3 0.0,E4 0.0,E5 0.0,E6 0.0}}
JPosSend_log[97]={cmdIdx 747289008,dt 0.0,cmdPos {A1 -106.622528,A2 -31.4800682,A3 -40.7959671,A4 -36.6705093,A5 72.0757370,A6 139.748947,E1 0.0,E2 0.0,E3 0.0,E4 0.0,E5 0.0,E6 0.0}}
JPosSend_log[98]={cmdIdx 747289030,dt 0.0,cmdPos {A1 -106.622528,A2 -31.4800682,A3 -40.7959671,A4 -36.6705093,A5 72.0757370,A6 139.748947,E1 0.0,E2 0.0,E3 0.0,E4 0.0,E5 0.0,E6 0.0}}
JPosSend_log[99]={cmdIdx 747289052,dt 0.0,cmdPos {A1 -106.622528,A2 -31.4800682,A3 -40.7959671,A4 -36.6705093,A5 72.0757370,A6 139.748947,E1 0.0,E2 0.0,E3 0.0,E4 0.0,E5 0.0,E6 0.0}}
JPosSend_log[100]={cmdIdx 747289074,dt 0.0,cmdPos {A1 -106.622528,A2 -31.4800682,A3 -40.7959671,A4 -36.6705093,A5 72.0757370,A6 139.748947,E1 0.0,E2 0.0,E3 0.0,E4 0.0,E5 0.0,E6 0.0}}


DECL CircQueue OpState_q={size 100,istart 100,iend 100}
DECL ROS_OpStateItem OpState_log[100]
OpState_log[1]={type #KRL_PTP,t_recv 1384537377}
OpState_log[2]={type #KRL_PTP,t_recv 1384540294}
OpState_log[3]={type #KRL_PTP,t_recv 1386205016}
OpState_log[4]={type #KRL_PTP,t_recv 1386206389}
OpState_log[5]={type #KRL_PTP,t_recv 1386559770}
OpState_log[6]={type #KRL_PTP,t_recv 1386561494}
OpState_log[7]={type #KRL_PTP,t_recv 1387364730}
OpState_log[8]={type #KRL_PTP,t_recv 1387366262}
OpState_log[9]={type #KRL_PTP,t_recv 1388423610}
OpState_log[10]={type #KRL_PTP,t_recv 1388425346}
OpState_log[11]={type #KRL_PTP,t_recv 1388606551}
OpState_log[12]={type #KRL_PTP,t_recv 1388607932}
OpState_log[13]={type #KRL_PTP,t_recv 324872595}
OpState_log[14]={type #KRL_PTP,t_recv 325083924}
OpState_log[15]={type #KRL_PTP,t_recv 326372804}
OpState_log[16]={type #KRL_PTP,t_recv 326373597}
OpState_log[17]={type #KRL_PTP,t_recv 334923797}
OpState_log[18]={type #KRL_PTP,t_recv 334928070}
OpState_log[19]={type #KRL_PTP,t_recv 349636356}
OpState_log[20]={type #KRL_PTP,t_recv 349639923}
OpState_log[21]={type #KRL_PTP,t_recv 14267474}
OpState_log[22]={type #KRL_PTP,t_recv 14269515}
OpState_log[23]={type #KRL_PTP,t_recv 22314607}
OpState_log[24]={type #KRL_PTP,t_recv 22316392}
OpState_log[25]={type #KRL_PTP,t_recv 334624858}
OpState_log[26]={type #KRL_PTP,t_recv 7687024}
OpState_log[27]={type #KRL_PTP,t_recv 182575304}
OpState_log[28]={type #KRL_PTP,t_recv 193102220}
OpState_log[29]={type #KRL_PTP,t_recv 194086568}
OpState_log[30]={type #KRL_PTP,t_recv 194550776}
OpState_log[31]={type #KRL_PTP,t_recv 354626651}
OpState_log[32]={type #KRL_PTP,t_recv 354628438}
OpState_log[33]={type #KRL_PTP,t_recv 2534088}
OpState_log[34]={type #KRL_PTP,t_recv 385044118}
OpState_log[35]={type #KRL_PTP,t_recv 385824798}
OpState_log[36]={type #KRL_PTP,t_recv 390734816}
OpState_log[37]={type #KRL_PTP,t_recv 393085856}
OpState_log[38]={type #KRL_PTP,t_recv 394148464}
OpState_log[39]={type #KRL_PTP,t_recv 394150384}
OpState_log[40]={type #KRL_PTP,t_recv 395730376}
OpState_log[41]={type #KRL_PTP,t_recv 395732357}
OpState_log[42]={type #KRL_PTP,t_recv 687210844}
OpState_log[43]={type #KRL_PTP,t_recv 687213254}
OpState_log[44]={type #KRL_PTP,t_recv 689153053}
OpState_log[45]={type #KRL_PTP,t_recv 689154981}
OpState_log[46]={type #KRL_PTP,t_recv 690849903}
OpState_log[47]={type #KRL_PTP,t_recv 690851573}
OpState_log[48]={type #KRL_PTP,t_recv 691807475}
OpState_log[49]={type #KRL_PTP,t_recv 691809294}
OpState_log[50]={type #KRL_PTP,t_recv 691994199}
OpState_log[51]={type #KRL_PTP,t_recv 691995967}
OpState_log[52]={type #KRL_PTP,t_recv 695355394}
OpState_log[53]={type #KRL_PTP,t_recv 695357560}
OpState_log[54]={type #KRL_PTP,t_recv 695504160}
OpState_log[55]={type #KRL_PTP,t_recv 695506343}
OpState_log[56]={type #KRL_PTP,t_recv 778672097}
OpState_log[57]={type #KRL_PTP,t_recv 778673914}
OpState_log[58]={type #KRL_PTP,t_recv 779328738}
OpState_log[59]={type #KRL_PTP,t_recv 779330347}
OpState_log[60]={type #KRL_PTP,t_recv 823172212}
OpState_log[61]={type #KRL_PTP,t_recv 823174655}
OpState_log[62]={type #KRL_PTP,t_recv 949794832}
OpState_log[63]={type #KRL_PTP,t_recv 949796983}
OpState_log[64]={type #KRL_PTP,t_recv 1014418153}
OpState_log[65]={type #KRL_PTP,t_recv 1014420325}
OpState_log[66]={type #KRL_PTP,t_recv 1016294953}
OpState_log[67]={type #KRL_PTP,t_recv 1016296853}
OpState_log[68]={type #KRL_PTP,t_recv 1017318121}
OpState_log[69]={type #KRL_PTP,t_recv 1017319805}
OpState_log[70]={type #KRL_PTP,t_recv 1017703815}
OpState_log[71]={type #KRL_PTP,t_recv 1017705773}
OpState_log[72]={type #KRL_PTP,t_recv 1040953719}
OpState_log[73]={type #KRL_PTP,t_recv 1040955638}
OpState_log[74]={type #KRL_PTP,t_recv 1543926500}
OpState_log[75]={type #KRL_PTP,t_recv 1543928972}
OpState_log[76]={type #RSI4ms_Pos,t_recv 1544046947}
OpState_log[77]={type #KRL_PTP,t_recv 1544073195}
OpState_log[78]={type #RSI4ms_Pos,t_recv 1544126677}
OpState_log[79]={type #RSI4ms_Pos,t_recv 1544158677}
OpState_log[80]={type #RSI4ms_Pos,t_recv 1544185519}
OpState_log[81]={type #KRL_PTP,t_recv 1544743688}
OpState_log[82]={type #KRL_PTP,t_recv 1544745762}
OpState_log[83]={type #RSI4ms_Pos,t_recv 1544788643}
OpState_log[84]={type #KRL_PTP,t_recv 1544849276}
OpState_log[85]={type #KRL_PTP,t_recv 1553083532}
OpState_log[86]={type #KRL_PTP,t_recv 1553085595}
OpState_log[87]={type #KRL_PTP,t_recv 405112059}
OpState_log[88]={type #KRL_PTP,t_recv 405114216}
OpState_log[89]={type #KRL_PTP,t_recv 473732823}
OpState_log[90]={type #KRL_PTP,t_recv 473734664}
OpState_log[91]={type #KRL_PTP,t_recv 736146806}
OpState_log[92]={type #KRL_PTP,t_recv 736148487}
OpState_log[93]={type #KRL_PTP,t_recv 737505135}
OpState_log[94]={type #KRL_PTP,t_recv 737506977}
OpState_log[95]={type #KRL_PTP,t_recv 738187113}
OpState_log[96]={type #KRL_PTP,t_recv 738189341}
OpState_log[97]={type #KRL_PTP,t_recv 745622801}
OpState_log[98]={type #KRL_PTP,t_recv 745624479}
OpState_log[99]={type #KRL_PTP,t_recv 746352895}
OpState_log[100]={type #KRL_PTP,t_recv 746354593}


DECL MODULEPARAM_T LAST_TP_PARAMS={PARAMS[] "Kuka.VelocityFieldEnabled=True; Kuka.ColDetectFieldEnabled=True; Kuka.MovementParameterFieldEnabled=True; Kuka.IsAngleEnabled=False; Kuka.PointName=drop4; Kuka.FrameData.base_no=0; Kuka.FrameData.tool_no=10; Kuka.FrameData.ipo_frame=#BASE; Kuka.FrameData.point2=; Kuka.isglobalpoint=False; Kuka.MoveDataPtpName=PDAT05; Kuka.MovementDataPdat.apo_mode=#CDIS; Kuka.MovementDataPdat.apo_dist=100; Kuka.MovementData.vel=20; Kuka.MovementData.acc=100; Kuka.MovementData.exax_ign=0; Kuka.VelocityPtp=20; Kuka.BlendingEnabled=False; Kuka.APXEnabled=False; Kuka.CurrentCDSetIndex=0; Kuka.MoveDataName=CPDAT1; Kuka.MovementData.cb={AUX_PT {ORI #CONSIDER,E1 #CONSIDER,E2 #CONSIDER,E3 #CONSIDER,E4 #CONSIDER,E5 #CONSIDER,E6 #CONSIDER},TARGET_PT {ORI #INTERPOLATE,E1 #INTERPOLATE,E2 #INTERPOLATE,E3 #INTERPOLATE,E4 #INTERPOLATE,E5 #INTERPOLATE,E6 #INTERPOLATE}}; Kuka.MovementData.apo_fac=50; Kuka.MovementData.apo_dist=500; Kuka.MovementData.axis_acc=100; Kuka.MovementData.axis_vel=100; Kuka.MovementData.circ_typ=#BASE; Kuka.MovementData.jerk_fac=50; Kuka.MovementData.ori_typ=#VAR; Kuka.VelocityPath=2  "}
DECL PDAT PPDAT05={VEL 20.0000,ACC 100.000,APO_DIST 100.000,APO_MODE #CDIS,GEAR_JERK 100.000,EXAX_IGN 0}
DECL FDAT Fdrop4={TOOL_NO 10,BASE_NO 0,IPO_FRAME #BASE,POINT2[] " "}
DECL E6POS Xdrop4={X 666666.688,Y 66.6000,Z 666.660,A 6.60000,B 66.6600,C 666.600,S 0,T 0,E1 0.0,E2 0.0,E3 0.0,E4 0.0,E5 0.0,E6 0.0}
ENDDAT
